FUNCTION_BLOCK FB_QualisysInterface
VAR_INPUT
END_VAR
VAR_OUTPUT
	bodyComponent : ST_RT6DComponent;
	markerComponent : ST_3DMarkerPositionNoLabelComponent;
	
	feedback : ST_FeedbackQualisys;
	
	active : BOOL := FALSE;
END_VAR
VAR
	// Udp related
	udpServer : FB_UdpServerRT(0, 0, 0, 0, 0); // Dummy constructor
	

	// Header 
	qrtPacket : ST_RTDataQRTPacket;
	qrtComponent : ARRAY [1..100] OF ST_RTComponentData;
	
	offset : UDINT;
	comp : UDINT;
	
	// HMi data
	pTxHmi : POINTER TO ST_TxHmiQualisys;
	
	// Actviity monitoring
	frame : DINT := 0;
	frameOld : DINT := 0;
	frameLoss : DINT := 0;
	
	stZero3DMarkerPositionNoLabelComponent : ST_3DMarkerPositionNoLabelComponent;
	
	// Marker tracking
	dMarker : REAL := 62.0;
	eMin : REAL;
	e : REAL;
	i : UDINT;
	j : UDINT;
	d : REAL;
	
	
	iSave : UDINT;
	jSave : UDINT;
	dSave : REAL;
	xSave : REAL;
	ySave : REAL;
	zSave : REAL;
	
	iMarker : ST_3DMarkerPositionNoLabel;
	jMarker : ST_3DMarkerPositionNoLabel;

END_VAR

// Check activity
frame := UDINT_TO_DINT(qrtPacket.nFramenumber);
IF frame <> frameOld THEN
	// Update frame old
	frameOld := frame;
	
	// Reset frameLoss
	frameLoss := 0;
ELSE
	// Count frame losses
	frameLoss := frameLoss + 1;
END_IF

// Set activity status after 1 second given 5ms in ms
IF frameLoss > 200 THEN
	active := FALSE;
ELSE
	active := TRUE;
END_IF

// Update HMI data
UpdateHMI();

// Exchange Udp data
udpServer();

// Decode Udp packet
MEMCPY(ADR(qrtPacket), ADR(udpServer.rxBuffer), SIZEOF(ST_RTDataQRTPacket));

// Zero out data
MEMCPY(ADR(markerComponent), ADR(stZero3DMarkerPositionNoLabelComponent), SIZEOF(ST_3DMarkerPositionNoLabelComponent));

offset := SIZEOF(ST_RTDataQRTPacket);
FOR comp := 1 TO qrtPacket.nComponentCount DO
	// Read components header
	MEMCPY(ADR(qrtComponent[comp]), ADR(udpServer.rxBuffer) + offset, SIZEOF(ST_RTComponentData));
	
	// Defoce components
	CASE qrtComponent[comp].nType OF
		1 : // 3D marker data 

		2 : // Unidentified 3D marker data
		MEMCPY(ADR(markerComponent), ADR(udpServer.rxBuffer) + offset, qrtComponent[comp].nSize); 
		
		3 : // Analog data from available analog devices
		
		4 : // Force data from available force plates.
		
		5 : // 6D data - position and rotation matrix
		MEMCPY(ADR(bodyComponent), ADR(udpServer.rxBuffer) + offset, qrtComponent[comp].nSize);
		
		6 : // 6D data - position and Euler angles
		
		7 : // 2D marker data
		
		8 : // Linearized 2D marker data
		
		9 : // 3D marker data with residuals
		
		10 : // Unidentified 3D marker data with residuals
		
		11 : // 6D data - position and rotation matrix with residuals
		
		12 : // 6D data - position and Euler angles with residuals
		
		13 : // Analog data from available analog devices
		
		14 : // Image frame from a specific camera
		
		15 : // Force data from available force plates
		
	END_CASE
	
	// Increment component byte offset
	offset := offset + SIZEOF(ST_RTComponentData) + qrtComponent[comp].nSize;
END_FOR

// Get hook position
IF active THEN
	IF markerComponent.nMarkers >= 2 THEN
		// Reset eMin to a default "high" value
		eMin := 1E10;
		
		FOR i := 0 TO markerComponent.nMarkers DO
			FOR j := 0 TO markerComponent.nMarkers DO
				// Calculate norm
				d := GetNorm(markerComponent.markers[i], markerComponent.markers[j]);
				e := ABS(d - dMarker);
				
				// Check if current marker set is closer than the others
				IF e < eMin THEN
					eMin := e;
					
					dSave := d;
					iSave := i;
					jSave := j;
				END_IF
			END_FOR
		END_FOR
		// Pick saved markers
		iMarker := markerComponent.markers[iSave];
		jMarker := markerComponent.markers[jSave];
		
		// Calculate average marker
		feedback.dist := dSave/1000.0;
		
		xSave := (iMarker.x + jMarker.x)/2.0;
		ySave := (iMarker.y + jMarker.y)/2.0;
		zSave := (iMarker.z + jMarker.z)/2.0;
		
	ELSIF markerComponent.nMarkers = 1 THEN
		// Indicate that hook is based on a single marker
		feedback.dist := 0.0;
		
		xSave := markerComponent.markers[0].x;
		ySave := markerComponent.markers[0].y;
		zSave := markerComponent.markers[0].z;
	ELSE	
		// Indicate that no markers are detected
		feedback.dist := -1.0;
	END_IF
	
	// mm -> m
	feedback.pos[0] := REAL_TO_LREAL(xSave/1000.0);
	feedback.pos[1] := REAL_TO_LREAL(ySave/1000.0);
	feedback.pos[2] := REAL_TO_LREAL(zSave/1000.0);
	
END_IF

METHOD FB_exit : BOOL
VAR_INPUT
	bInCopyCode : BOOL; // if TRUE, the exit method is called for exiting an instance that is copied afterwards (online change).
END_VAR
END_METHOD

METHOD FB_init : BOOL
VAR_INPUT
	bInitRetains : BOOL; // if TRUE, the retain variables are initialized (warm start / cold start)
	bInCopyCode : BOOL;  // if TRUE, the instance afterwards gets moved into the copy code (online change)

	// Init variables
	_localPort : UINT;
	_pTxHmi : POINTER TO ST_TxHmiQualisys;
END_VAR
// Initilize the udpServer
udpServer.FB_init(
	bInitRetains,
	bInCopyCode,
	_localPort,
	0,
	0,
	0,
	0
);

pTxHmi := _pTxHmi;
END_METHOD

METHOD FB_reinit : BOOL
VAR_INPUT
END_VAR
END_METHOD

METHOD PRIVATE GetNorm : REAL
VAR_INPUT
	m1 : ST_3DMarkerPositionNoLabel;
	m2 : ST_3DMarkerPositionNoLabel;
END_VAR

VAR
	x : REAL;
	y : REAL;
	z : REAL;
END_VAR
// Vector 
x := m2.x - m1.x;
y := m2.y - m1.y;
z := m2.z - m1.z;

// Norm
GetNorm := SQRT(x*x + y*y + z*z);
END_METHOD

METHOD PRIVATE UpdateHMI : BOOL
VAR_INPUT
END_VAR

VAR
	i : UDINT;
END_VAR
// Update global Hmi data
IF active THEN
	pTxHmi^.status := 0;
ELSE
	pTxHmi^.status := -1;
END_IF

// Update feedback data
pTxHmi^.dist := LREAL_TO_REAL(feedback.dist);
pTxHmi^.x := LREAL_TO_REAL(feedback.pos[0]);
pTxHmi^.y := LREAL_TO_REAL(feedback.pos[1]);
pTxHmi^.z := LREAL_TO_REAL(feedback.pos[2]);

// Marker data
FOR i := 0 TO 9 DO
	pTxHmi^.markers[i] := markerComponent.markers[i];
END_FOR
END_METHOD

END_FUNCTION_BLOCK

(* stored: Version 1.1.0.1, ProductVersion 3.1.4022.18
   POU FB_QualisysInterface: Id {314e7cd5-278b-4ae6-86cd-8f8bb2148757}, SpecialFunc None
   Method FB_exit: Id {218c743a-0e42-4699-b90a-ee85a516329b}
   Method FB_init: Id {f7454e96-6d71-45e3-a8c8-afff39670148}
   Method FB_reinit: Id {a77f1cd7-b4fd-4175-afb3-b8ab028ade9c}
   Method GetNorm: Id {728830f4-0a5a-4307-8c1f-0576f2b3aab7}
   Method UpdateHMI: Id {90c4b41f-ef66-41d0-8737-7df7866b25e1} *)
